// TwinCAT 3 PLC project SuperviserPLC
// ProgramVersion: 3.1.4026.20
// libraries:
//   Tc2_Standard, * (Beckhoff Automation GmbH)
//   Tc2_System, * (Beckhoff Automation GmbH)
//   Tc2_TcpIp, * (Beckhoff Automation GmbH)
//   Tc2_Utilities, * (Beckhoff Automation GmbH)
//   Tc3_EventLogger, * (Beckhoff Automation GmbH)
//   Tc3_JsonXml, * (Beckhoff Automation GmbH)
//   Tc3_Module, * (Beckhoff Automation GmbH)
// project tree:
//   Navitrol Supervisor/Common types/ ST_SectionHeader.TcDUT (not stored), ST_SupervisorHeader.TcDUT
//   Navitrol Supervisor/ FB_Supervisor.TcPOU
//   Navitrol Supervisor/Navitrol to Supervisor response/1100/ ST_1100_Position_initialization_started.TcDUT
//   Navitrol Supervisor/Navitrol to Supervisor response/1101/Components/ E_1101_Initialization_result.TcDUT
//   Navitrol Supervisor/Navitrol to Supervisor response/1101/ ST_1101_Position_initialized.TcDUT (not stored)
//   Navitrol Supervisor/Navitrol to Supervisor response/1126/Components/ ST_1126_Omni_wheels_ref_struct.TcDUT, ST_1126_Supervisor_status_out.TcDUT
//   Navitrol Supervisor/Navitrol to Supervisor response/1126/ ST_1126_Motor_control_omni_response.TcDUT (not stored)
//   Navitrol Supervisor/Navitrol to Supervisor response/3102/Components/ E_3102_Error_status.TcDUT (not stored), E_3102_Position_initialize_status.TcDUT (not stored), E_3102_State.TcDUT (not stored)
//   Navitrol Supervisor/Navitrol to Supervisor response/3102/Components/Sections/1/ ST_3102_1_General_section.TcDUT
//   Navitrol Supervisor/Navitrol to Supervisor response/3102/ ST_3102_Navitrol_status.TcDUT
//   Navitrol Supervisor/Navitrol to Supervisor response/ Param_Supervisor_response.TcGVL (not stored), U_Recived_bytes_from_Navitrol.TcDUT (not stored)
//   Navitrol Supervisor/Supervisor to Navitrol message/1001/ ST_1001_Initialize_position.TcDUT (not stored)
//   Navitrol Supervisor/Supervisor to Navitrol message/1026/Components/ E_1026_Set_drive_mode.TcDUT (not stored), ST_1026_Omni_wheels_struct.TcDUT (not stored), ST_1026_Supervisor_status_bits.TcDUT (not stored)
//   Navitrol Supervisor/Supervisor to Navitrol message/1026/ ST_1026_Measurement_update_generic_omni_drive.TcDUT
//   Navitrol Supervisor/Supervisor to Navitrol message/3002/Components/ E_3002_Set_ESTOP.TcDUT (not stored), E_3002_Status.TcDUT
//   Navitrol Supervisor/Supervisor to Navitrol message/3002/Components/Sections/2/Components/ E_3002_2_Enable_manual_control.TcDUT, E_3002_2_Inactive_Active.TcDUT (not stored)
//   Navitrol Supervisor/Supervisor to Navitrol message/3002/Components/Sections/2/ ST_3002_2_Manual_section.TcDUT (not stored)
//   Navitrol Supervisor/Supervisor to Navitrol message/3002/Components/Sections/6/Components/ E_3002_6_Joystick1_control_mode.TcDUT, E_3002_6_Joystick2_control_mode.TcDUT (not stored), E_3002_6_Steer_type_selection.TcDUT
//   Navitrol Supervisor/Supervisor to Navitrol message/3002/Components/Sections/6/ ST_3002_6_Remote_control_section.TcDUT
//   Navitrol Supervisor/Supervisor to Navitrol message/3002/Components/Sections/8/Components/ ST_3002_8_Binary_data.TcDUT, ST_3002_8_Error_status.TcDUT (not stored)
//   Navitrol Supervisor/Supervisor to Navitrol message/3002/Components/Sections/8/ ST_3002_8_Battery_section.TcDUT
//   Navitrol Supervisor/Supervisor to Navitrol message/3002/Components/Sections/ F_SetSectionHeaderInfo.TcPOU
//   Navitrol Supervisor/Supervisor to Navitrol message/3002/ ST_3002_Supervisor_Status.TcDUT
//   Navitrol Supervisor/Supervisor to Navitrol message/ F_SetHeaderInfo.TcPOU (not stored)
//   / PlcTask.TcTTO
//   POUs/ MAIN.TcPOU
// real-time tasks:
//   TASK PlcTask: cycle T#1ms, priority 20, ADS port 350
// motion (NC):
//   TASK NC-Task 1 SAF: cycle T#2ms, priority 4, ADS port 501
//   TASK NC-Task 1 SVB: cycle T#10ms, priority 8, ADS port 511
//   AXIS LeftWheel (id 1)
//     General: UnitName=m
//     Dynamic: AccelerationMaximum=1, DecelerationMaximum=1, Acceleration=2222, Deceleration=2222, Jerk=224422000
//     Velo: SlowManual=0.6, FastManual=1, Maximum=2.2
//     OtherSettings: AllowMotionCmdToSlave=true
//     encoder EncType=1
//       EncPara: ScaleFactorNumerator=1e-07, EncMode=3
//     drive DrvType=5
//       Analog: VeloReferenz=2.2, TorqueSetpointScale=10, ScaleFactorActTorque=0.1
//       TimeComp: TaskDelayCycles=1
//     controller CtrType=1
//       CtrPara: PriorControlFactor=1
//         Observer: BandWidth=20
//   AXIS RightWheel (id 2)
//     General: UnitName=m
//     Dynamic: AccelerationMaximum=1, DecelerationMaximum=1, Acceleration=2222, Deceleration=2222, Jerk=224422000
//     Velo: SlowManual=0.6, FastManual=1, Maximum=2.2
//     OtherSettings: AllowMotionCmdToSlave=true
//     encoder EncType=1
//       EncPara: ScaleFactorNumerator=1e-07, EncMode=3
//     drive DrvType=5
//       Analog: VeloReferenz=2.2, TorqueSetpointScale=10, ScaleFactorActTorque=0.1
//       TimeComp: TaskDelayCycles=1
//     controller CtrType=1
//       CtrPara: PriorControlFactor=1
//         Observer: BandWidth=20
// variable links:
//   SupervisorPLC Instance <-> NC-Task 1 SAF/Axes/LeftWheel
//     PlcTask Inputs/MAIN.LeftWheel.NcToPlc <-> Outputs/ToPlc
//     PlcTask Outputs/MAIN.LeftWheel.PlcToNc <-> Inputs/FromPlc
//   SupervisorPLC Instance <-> NC-Task 1 SAF/Axes/RightWheel
//     PlcTask Inputs/MAIN.RightWheel.NcToPlc <-> Outputs/ToPlc
//     PlcTask Outputs/MAIN.RightWheel.PlcToNc <-> Inputs/FromPlc

CONFIGURATION SuperviserPLC
    RESOURCE PLC ON TwinCAT3
        TASK PlcTask(INTERVAL := T#1ms, PRIORITY := 20);
        PROGRAM MAIN WITH PlcTask : MAIN;
    END_RESOURCE
END_CONFIGURATION

// ---- Navitrol Supervisor/Common types/ST_SupervisorHeader.TcDUT
{attribute 'pack_mode' := '1'}
{attribute 'hide_all_locals'}
TYPE ST_SupervisorHeader :
	STRUCT
		Protocol_version : UINT;	
		Message_ID		 : UINT;
		Message_length	 : UDINT;
	END_STRUCT
END_TYPE
//When sending a message from Supervisor to Navitrol, this is populated using F_SetHeaderInfo.

// ---- Navitrol Supervisor/Navitrol to Supervisor response/1100/ST_1100_Position_initialization_started.TcDUT
{attribute 'pack_mode' := '1'}
TYPE ST_1100_Position_initialization_started EXTENDS ST_SupervisorHeader :
STRUCT
END_STRUCT
END_TYPE

// ---- Navitrol Supervisor/Navitrol to Supervisor response/1101/Components/E_1101_Initialization_result.TcDUT
{attribute 'qualified_only'}
{attribute 'strict'}
{attribute 'to_string'}
TYPE E_1101_Initialization_result : (
		Failure := 0,
		Success := 1
	) UINT;
END_TYPE
//0 - Failure
//	The position initialization can fail for example if
//		- A good position is not found within pos_ini_max_d..-parameters from the given pos init point
//		- A good position is not found within value of pos_init_max_wait_time-parameter
//		- The AGV is not stationary state, it is performing load or there are scanner related errors active.
//1 - Success
//		- A good position was found near the given position initialization point and position was successfully initialized.

// ---- Navitrol Supervisor/Navitrol to Supervisor response/1126/Components/ST_1126_Omni_wheels_ref_struct.TcDUT
{attribute 'pack_mode' := '1'}
TYPE ST_1126_Omni_wheels_ref_struct :
	STRUCT
		Steer_angle_reference : REAL;
		Wheel_speed_reference : REAL;
	END_STRUCT
END_TYPE

// ---- Navitrol Supervisor/Navitrol to Supervisor response/1126/Components/ST_1126_Supervisor_status_out.TcDUT
{attribute 'pack_mode' := '1'}
TYPE ST_1126_Supervisor_status_out :
	STRUCT
		Navitrol_error : BIT; //	Navitrol has ANY error active AND is unable TO drive.
		Reserved_1	   : BIT;
		Reserved_2	   : BIT;
		Reserved_3	   : BIT;
		Reserved_4	   : BIT;
		Reserved_5	   : BIT;
		Reserved_6	   : BIT;
		Brake_release  : BIT;  //	Navitrol requests Supevisor to release brakes to start driving
		Reserved	   : BYTE; //	Not in use	
	END_STRUCT
END_TYPE

// ---- Navitrol Supervisor/Navitrol to Supervisor response/3102/Components/Sections/1/ST_3102_1_General_section.TcDUT
{attribute 'pack_mode' := '1'}
TYPE ST_3102_1_General_section EXTENDS ST_SectionHeader :
	STRUCT
		Battery_voltage : REAL; // V
		On_route		: UINT; // 1 on route, 0 not on route
	END_STRUCT
END_TYPE

// ---- Navitrol Supervisor/Navitrol to Supervisor response/3102/ST_3102_Navitrol_status.TcDUT
{attribute 'pack_mode' := '1'}
TYPE ST_3102_Navitrol_status EXTENDS ST_SupervisorHeader :
	STRUCT
		DefaultSectionLength	   : UDINT;
		State					   : E_3102_State;
		X_coordinate			   : REAL; //In meters
		Y_coordinate			   : REAL; //In meters
		Heading					   : REAL; //Radians
		Level					   : DINT; //Level ID
		Speed					   : REAL; //m/s
		Position_initialize_status : E_3102_Position_initialize_status;
		Position_confidence		   : UINT; //Position confidence in percentage (1 - 100%)
		Error_status			   : E_3102_Error_status;
		//Additional sections can be added bellow - based on what is requested in the array "Section_IDs" in ST_3002_Supervisor_Status.
		General_section			   : ST_3102_1_General_section;
	END_STRUCT
END_TYPE

// ---- Navitrol Supervisor/Supervisor to Navitrol message/1026/ST_1026_Measurement_update_generic_omni_drive.TcDUT
{attribute 'pack_mode' := '1'}
TYPE ST_1026_Measurement_update_generic_omni_drive EXTENDS ST_SupervisorHeader :
	STRUCT
		Message_number	  : UDINT;
		Set_drive_mode	  : E_1026_Set_drive_mode;
		Supervisor_status : ST_1026_Supervisor_status_bits := (Brake_released := TRUE);
		Number_of_wheels  : UINT						   := 2;
	Omni_wheels: ARRAY [0..1] OF ST_1026_Omni_wheels_struct := [2((Steer_angle := 0.1))];		
	END_STRUCT
END_TYPE

// ---- Navitrol Supervisor/Supervisor to Navitrol message/3002/Components/E_3002_Status.TcDUT
{attribute 'qualified_only'}
{attribute 'strict'}
{attribute 'to_string'}
TYPE E_3002_Status : (
		Not_ok := 0, //ERROR_PLC_FAILURE will be activated, and additionally manual driving will be prevented.
		Ok	   := 1	 //Navitrol is allowed to drive the AGV.
	) UINT;
END_TYPE

// ---- Navitrol Supervisor/Supervisor to Navitrol message/3002/Components/Sections/2/Components/E_3002_2_Enable_manual_control.TcDUT
{attribute 'qualified_only'}
{attribute 'strict'}
{attribute 'to_string'}
TYPE E_3002_2_Enable_manual_control : (
		Enable_control	:= 0,
		Disable_control := 1
	) UINT;
END_TYPE

(*
Used to enable manual control from this section:
	0 - Enable control
Navitrol will activate manual mode and sets WARNING_ETH_MANUAL_MODE. This section can be used to drive the AGV.
	1 - Disable control
Navitrol will ignore any controls from this section.
*)

// ---- Navitrol Supervisor/Supervisor to Navitrol message/3002/Components/Sections/6/Components/E_3002_6_Joystick1_control_mode.TcDUT
{attribute 'qualified_only'}
{attribute 'strict'}
{attribute 'to_string'}
TYPE E_3002_6_Joystick1_control_mode : (
		No_control	   := 0,
		Old_control	   := 1,
		Vector_control := 2
	)UINT;
END_TYPE

(*
Selects the joystick 1 control mode:
	0 - No control
Joystick 1 x and y values are ignored.
	1 - Old control
	Not recommended
	Navitrol activates manual mode. Curvature is calculated directly from joystick 1 x value and the speed from joystick 1 y value.
2 - Vector control
	Recommended
	Navitrol activates manual mode. A unit vector is calculated from joystick 1 xy-values. The speed comes from the length of the vector (Positive when y is positive) and the curvature from its angle from the Y-axis.
	For example AGV drives forward and curves right when x and y are positive.
	For more information, see "Joystick System" chapter from Web Interface document

*)

// ---- Navitrol Supervisor/Supervisor to Navitrol message/3002/Components/Sections/6/Components/E_3002_6_Steer_type_selection.TcDUT
{attribute 'qualified_only'}
{attribute 'strict'}
{attribute 'to_string'}
TYPE E_3002_6_Steer_type_selection : (
		Invalid					:= 0,
		Front_wheel_steer		:= 1,
		Mid_wheel_steer			:= 2,
		Rear_wheel_steer		:= 3,
		Pivot_steer				:= 5,
		Parallel_steer_forward	:= 6,
		Parallel_steer_backward := 7
	);
END_TYPE

(*
1 - Front wheel steer
Only for omni drives. Moves the navigation point to between the front wheels. With this steer type almost all turning control will be done by the rear wheels.
2 - Mid wheel steer
	Normal driving. The normal navigation point is used.
3 - Rear wheel steer
	Only for omni drives. Moves the navigation point to between the rear wheels. With this steer type almost all turning control will be done by the front wheels.
5 - Pivot steer
	Pivot curvature is always given, and supervisor can control only the speed up to maximum of pivot_speed-parameter. This mode should only be activated, if the AGV can pivot.
6 - Parallel steer forward
	Only for omni drives.
	The curvature in this mode is always zero. Instead of curvature supervisor controls the frame heading instead and speed. Wheels will rotate forward with positive speed reference.
7 - Parallel steer backward
	Only for omni drives.
	The curvature in this mode is always zero. Instead of curvature supervisor controls the frame heading instead and speed. Wheels will rotate backwards with positive speed reference.

*)

// ---- Navitrol Supervisor/Supervisor to Navitrol message/3002/Components/Sections/6/ST_3002_6_Remote_control_section.TcDUT
{attribute 'pack_mode' := '1'}
TYPE ST_3002_6_Remote_control_section EXTENDS ST_SectionHeader :
	STRUCT
		Joystick1_control_mode : E_3002_6_Joystick1_control_mode;
		Joystick1_x			   : REAL;
		Joystick1_y			   : REAL;
		Joystick2_control_mode : E_3002_6_Joystick2_control_mode;
		Joystick2_x			   : REAL; //0 - Not in use
		Joystick2_y			   : REAL; (*Lift actuator height reference control.
										If the given y-value is larger than 0.1 actuator control is enabled. 
										And the y-value is scaled with actuator_eth_ctrl_scale-parameter and added to the previous actuator reference. 
										The actuator reference can be controlled only between values of actuator_min_val and actuator_max_val parameters.Valid values [-1...1]*)
		Steer_type_selection : E_3002_6_Steer_type_selection;
	END_STRUCT
END_TYPE

// ---- Navitrol Supervisor/Supervisor to Navitrol message/3002/Components/Sections/8/Components/ST_3002_8_Binary_data.TcDUT
{attribute 'pack_mode' := '1'}
TYPE ST_3002_8_Binary_data :
STRUCT
	Request_charge   : BIT; // This charge request info is show in motor control messages and in Navitrol battery status section if charging_cmd_source-parameter is set to 3. No drive orders or other actions are made based on this.
	Charging_active  : BIT; // Informs Navitrol that charging is active. Navitrol will set soft stop (parameter charging_prevents_driving).
	Balancing_active : BIT; // Informs Navitrol that battery balancing is active at charger. Navitrol will set soft stop (parameter charging_prevents_driving).
	Reserved_3       : BIT; // 0 - Not in use
	Reserved_4       : BIT; // 0 - Not in use
	Reserved_5       : BIT; // 0 - Not in use
	Reserved_6       : BIT; // 0 - Not in use
	Reserved_7       : BIT; // 0 - Not in use
END_STRUCT
END_TYPE

// ---- Navitrol Supervisor/Supervisor to Navitrol message/3002/Components/Sections/8/ST_3002_8_Battery_section.TcDUT
{attribute 'pack_mode' := '1'}
TYPE ST_3002_8_Battery_section EXTENDS ST_SectionHeader :
	STRUCT
		// Battery state of charge percentage. Valid values [0...100] 65535 - Not available

		// This will be used for determining the battery level if battery_percentage_from_mot_ctrl-parameter is set to 1.
		State_of_charge : UINT := 100;
		// Battery voltage in 0.1 Volts. For example, 4.2V would be 42 65535 - Not available

		// This will be used for determining the battery level if battery_percentage_from_mot_ctrl-parameter is set to 0.
		Voltage : UINT := 42;
		// Charge current / current draw in 0.1 Amperes. Negative values when battery is discharging

		// and positive values when battery is being charged. 32767 - Not available

		// Only for statistics - visible in Navitrol Monitor.
		Charge_current_draw : INT := 10;
		// Energy draw in 0.1 Ampere hours Negative values when battery is discharging

		// and positive values when battery is being charged. 32767 - Not available

		// Only for statistics - visible in Navitrol Monitor.
		Energy_draw : INT := 100;
		// Estimated time left in minutes until the battery is empty. 65535 - Not available

		// Only for statistics - visible in Navitrol Monitor.
		Time_remaining : UINT := 45;
		// Battery state of health percentage. Describes the overall state of the battery. Valid values [0...100] 65535 - Not available

		// Only for statistics - visible in Navitrol Monitor.
		State_of_health : UINT := 100;
		// Battery temperature in Celsius degrees. 32767 - Not available

		// Used to trigger WARNING_BATTERY_HIGH_TEMPERATURE if given temperature is larger than

		// battery_high_temperature_warning_limit_C and ERROR_BATTERY_HIGH_TEMPERATURE if larger

		// than battery_high_temperature_error_limit_C
		Temperature : INT := 32;
		// Total number of load cycles performed for the battery. 65535 - Not available

		// Only for statistics - visible in Navitrol Monitor.
		Load_cycle_count : UINT := 20;
		// Total number of operating hours of the battery. 65535 - Not available

		// Only for statistics - visible in Navitrol Monitor.
		Operating_hours : UINT := 155;
		// Voltage of the charger in 0.1 Volts. 65535 - Not available

		// Only for statistics - visible in Navitrol Monitor.
		Charger_voltage : UINT := 420;
		// Error status information. If any of the errors marked with * are active Navitrol Monitor will view its description

		// and Navitrol set WARNING_BATTERY_ERROR_OR_WARNING_ACTIVE 0 - No error
		Error_status : ST_3002_8_Error_status;
		// Battery related binary data and requests 0 - Inactive
		Binary_data : ST_3002_8_Binary_data;
		// 0 - Not in use
		Reserved : BYTE;
	END_STRUCT
END_TYPE

// ---- Navitrol Supervisor/Supervisor to Navitrol message/3002/ST_3002_Supervisor_Status.TcDUT
{attribute 'pack_mode' := '1'}
TYPE ST_3002_Supervisor_Status EXTENDS ST_SupervisorHeader :
	STRUCT
		Status			   : E_3002_Status := E_3002_Status.Ok;
		Set_Estop		   : E_3002_Set_ESTOP;
		Number_of_sections : UINT				 := 1;	 //Number of sections requested in response message 3102 - Needs to be the same number as the array size Section_IDs. if 0 - then Section_IDs can be commented out
		Section_IDs		   : ARRAY[0..0] OF UINT := [1]; //List of sections to send in the response message 3102
		Manual_section: ST_3002_2_Manual_section := (Enable_manual_control := E_3002_2_Enable_manual_control.Disable_control);		
		Battery_section	   : ST_3002_8_Battery_section;
	END_STRUCT
END_TYPE

// ---- POUs/MAIN.TcPOU
PROGRAM MAIN
VAR
	Supervisor				 : FB_Supervisor := (RemoteHost := '127.0.0.1', RemotePort := 2000);
END_VAR

Supervisor(Execute := TRUE);

END_PROGRAM

// ---- Navitrol Supervisor/FB_Supervisor.TcPOU
FUNCTION_BLOCK FB_Supervisor
VAR_INPUT
	RemoteHost									 : T_IPv4Addr := '127.0.0.1';
	RemotePort									 : UDINT	  := 2000;	  //Needs to match Navitrol parameter "supervisor_eth_port"
	CycleTime3002								 : TIME		  := T#100MS; //maximum interval 1 second
	CycleTime1026								 : TIME		  := T#30MS;  //This needs to match the Navitrol parameter "control_interval_us"
	Execute										 : BOOL;				  //Connect to Navitrol, and establish comuncations. If false, the socket is closed.
	st3002_Supervisor_Status					 : ST_3002_Supervisor_Status;
	st1026_Measurement_update_generic_omni_drive : ST_1026_Measurement_update_generic_omni_drive;
	Initialize_position							 : BOOL; //Rising edge trigger to send a Initialize position command 
	st1001_Initialize_position					 : ST_1001_Initialize_position := (X := 100.0, Y := 150.0);
END_VAR

VAR_OUTPUT
	st3102_Navitrol_status			   : ST_3102_Navitrol_status;
	st1126_Motor_control_omni_response : ST_1126_Motor_control_omni_response;
	st1101_Position_initialized		   : ST_1101_Position_initialized;
	Busy							   : BOOL;
	Error							   : BOOL;
	ErrorID							   : UDINT;
END_VAR

VAR
	State : (INIT_FBs,
		CLOSE_OLD_SOCKETS,
		CONNECT_TO_Server,
		COMS_ACTIVE,
		CLOSE_CONNECTION);
	CloseAll : FB_SocketCloseAll;
	Connect	 : FB_SocketConnect;
	Close	 : FB_SocketClose;

	//Event logging
	FirstScan  : BOOL := TRUE;
	ErrorMsg   : FB_TcMessage;
	WarnMsg	   : FB_TcMessage;
	VerboseMsg : FB_TcMessage;
END_VAR

IF FirstScan THEN
	ErrorMsg.CreateEx(stEventEntry := TC_EVENTS.TcpIpComms.ErrorMsg, ipSourceInfo := 0);
	VerboseMsg.CreateEx(stEventEntry := TC_EVENTS.TcpIpComms.VerboseMsg, ipSourceInfo := 0);
	WarnMsg.CreateEx(stEventEntry := TC_EVENTS.TcpIpComms.WarnMsg, ipSourceInfo := 0);
	FirstScan := FALSE;
END_IF

CASE State OF
	INIT_FBs:
		CloseAll(bExecute := FALSE);
		Connect(bExecute := FALSE);
		Close(bExecute := FALSE);
		Busy := FALSE;
		IF Execute THEN
			Busy := TRUE;
			IF CycleTime3002 = T#0S OR CycleTime3002 > T#1S THEN
				ErrorMsg.ipArguments.Clear().AddString('Invalid input CycleTime3002');
				ErrorMsg.Send();
				Error := TRUE;
				RETURN;
			END_IF

			State := CLOSE_OLD_SOCKETS;
			Error := FALSE;
			VerboseMsg.ipArguments.Clear().AddString('Starting communications to:').AddString(RemoteHost).AddUDInt(RemotePort);
			VerboseMsg.Send();
		END_IF

	CLOSE_OLD_SOCKETS: //In the event of online change or download
		CloseAll(sSrvNetId := '', bExecute := TRUE, tTimeout := T#10S);
		IF NOT CloseAll.bBusy THEN
			CloseAll(bExecute := FALSE);
			State := CONNECT_TO_Server;
		END_IF

	CONNECT_TO_Server:
		Connect(sSrvNetId	:= '',
				sRemoteHost := RemoteHost,
				nRemotePort := RemotePort,
				bExecute	:= TRUE,
				tTimeout	:= T#4S);

		IF NOT Connect.bBusy THEN
			IF NOT Connect.bError THEN
				IF Connect.hSocket.handle <> 0 THEN
					State := COMS_ACTIVE;
					VerboseMsg.ipArguments.Clear().AddString('Connected to server:').AddString(RemoteHost).AddUDInt(RemotePort).AddString('Local port').AddUDInt(Connect.hSocket.localAddr.nPort);
					VerboseMsg.Send();
				END_IF
			ELSE
				Error := TRUE;
				State := INIT_FBs;
				ErrorMsg.ipArguments.Clear().AddString('Failed to connect to server:').AddString(RemoteHost).AddUDInt(RemotePort).AddString(', Error:').AddUDInt(Connect.nErrId);
				ErrorMsg.Send();
			END_IF

			Connect(bExecute := FALSE);
		END_IF

	COMS_ACTIVE:
		SendMsg3002();
		SendMsg1026();
		SendMsg1001();
		ReciveAllMsgsAndParse();
		IF NOT Execute THEN
			VerboseMsg.ipArguments.Clear().AddString('Connection closed by user');
			VerboseMsg.Send();
			State := CLOSE_CONNECTION;
		END_IF

	CLOSE_CONNECTION:
		Close(sSrvNetId := '',
			  hSocket	:= Connect.hSocket,
			  bExecute	:= TRUE,
			  tTimeout	:= T#4S);

		IF NOT Close.bBusy THEN
			Close(bExecute := FALSE);
			State := INIT_FBs;
		END_IF
END_CASE

METHOD INTERNAL ReciveAllMsgsAndParse : HRESULT
VAR_INST
	Receive								   : FB_SocketReceive;
	ReceiveBuffer						   : U_Recived_bytes_from_Navitrol;
	NumOf1100MsgRecived					   : UDINT;
	st1100_Position_initialization_started : ST_1100_Position_initialization_started;
	NumOf1101MsgRecived					   : UDINT;
	NumOf3102MsgRecived					   : UDINT;
	NumOf1126MsgRecived					   : UDINT;
	UnknowMsgRecivedCounter				   : UDINT;
	UnknowMsg							   : U_Recived_bytes_from_Navitrol;
END_VAR
Receive(sSrvNetId := '',
		hSocket	  := Connect.hSocket,
		cbLen	  := SIZEOF(ReceiveBuffer),
		pDest	  := ADR(ReceiveBuffer),
		bExecute  := TRUE,
		tTimeout  := T#10S);

IF NOT Receive.bBusy THEN
	IF Receive.nRecBytes <> 0 THEN
		IF Receive.nRecBytes = SIZEOF(ReceiveBuffer) THEN
			ErrorMsg.ipArguments.Clear().AddString('Recive buffer is not large enough! Please increase the size of "Param_Supervisor_response.RecivedBytesBufferSize');
			ErrorMsg.Send();
			State	:= CLOSE_CONNECTION;
			Error	:= TRUE;
			ErrorID := Global.TC_EVENTS.TcGeneralAdsEventClass.NoMemory.nEventId;
			RETURN;
		END_IF

		CASE ReceiveBuffer.Header.Message_ID OF //Check what message type is being recived - then copy it into the correct structure
			1100:
				NumOf1100MsgRecived := NumOf1100MsgRecived + 1;
				MEMCPY(destAddr := ADR(st1100_Position_initialization_started), srcAddr := ADR(ReceiveBuffer), n := SIZEOF(st1100_Position_initialization_started));
				VerboseMsg.ipArguments.Clear().AddString('Position initialization started');
				VerboseMsg.Send();

			1101:
				NumOf1101MsgRecived := NumOf1101MsgRecived + 1;
				MEMCPY(destAddr := ADR(st1101_Position_initialized), srcAddr := ADR(ReceiveBuffer), n := SIZEOF(st1101_Position_initialized));
				VerboseMsg.ipArguments.Clear().AddString('Position initialization finished');
				VerboseMsg.Send();

			1126:
				NumOf1126MsgRecived := NumOf1126MsgRecived + 1;
				MEMCPY(destAddr := ADR(st1126_Motor_control_omni_response), srcAddr := ADR(ReceiveBuffer), n := SIZEOF(st1126_Motor_control_omni_response));

			3102:
				NumOf3102MsgRecived := NumOf3102MsgRecived + 1;
				MEMCPY(destAddr := ADR(st3102_Navitrol_status), srcAddr := ADR(ReceiveBuffer), n := SIZEOF(st3102_Navitrol_status));

		ELSE
			UnknowMsgRecivedCounter := UnknowMsgRecivedCounter + 1;
			MEMCPY(destAddr := ADR(UnknowMsg), srcAddr := ADR(ReceiveBuffer), n := SIZEOF(UnknowMsg));
			WarnMsg.ipArguments.Clear().AddString('Unknow msg type recived with ID:').AddUInt(ReceiveBuffer.Header.Message_ID).AddString('Contents:').AddBlob(pData := ADR(ReceiveBuffer), cbData := TO_UINT(Receive.nRecBytes));
			WarnMsg.Send();
		END_CASE
	END_IF

	Receive(bExecute := FALSE);

	//Clear recive buffer
	MEMSET(destAddr := ADR(ReceiveBuffer), fillByte := 0, n := SIZEOF(ReceiveBuffer));
END_IF

IF Receive.bError THEN
	ErrorMsg.ipArguments.Clear().AddString('Failed to Receive, Error:').AddUDInt(Receive.nErrId);
	ErrorMsg.Send();
	State	:= CLOSE_CONNECTION;
	Error	:= TRUE;
	ErrorID := Receive.nErrId;
END_IF
END_METHOD

METHOD INTERNAL SendMsg1001 : HRESULT
VAR_INST
	rtInitialize_position : R_TRIG;
	Send1001			  : FB_SocketSend;
END_VAR
rtInitialize_position(CLK := Initialize_position);
IF rtInitialize_position.Q THEN
	F_SetHeaderInfo(st1001_Initialize_position);
	MEMSET(destAddr := ADR(st1101_Position_initialized), fillByte := 0, n := SIZEOF(st1101_Position_initialized)); //Clear old results
END_IF

Send1001(sSrvNetId := '',
		 hSocket   := Connect.hSocket,
		 cbLen	   := SIZEOF(st1001_Initialize_position),
		 pSrc	   := ADR(st1001_Initialize_position),
		 bExecute  := rtInitialize_position.Q,
		 tTimeout  := T#2S);

IF Send1001.bError THEN
	ErrorMsg.ipArguments.Clear().AddString('Failed to send 1001 Error:').AddUDInt(Send1001.nErrId);
	ErrorMsg.Send();
END_IF
END_METHOD

METHOD INTERNAL SendMsg1026 : HRESULT
VAR_INST
	Timer1026 : TON;
	Send1026  : FB_SocketSend;
END_VAR
Timer1026(IN := NOT Timer1026.Q, PT := CycleTime1026);
IF Timer1026.Q THEN
	F_SetHeaderInfo(st1026_Measurement_update_generic_omni_drive);
	st1026_Measurement_update_generic_omni_drive.Message_number := st1026_Measurement_update_generic_omni_drive.Message_number + 1;
END_IF

Send1026(sSrvNetId := '',
		 hSocket   := Connect.hSocket,
		 cbLen	   := SIZEOF(st1026_Measurement_update_generic_omni_drive),
		 pSrc	   := ADR(st1026_Measurement_update_generic_omni_drive),
		 bExecute  := Timer1026.Q,
		 tTimeout  := T#2S);

IF Send1026.bError THEN
	ErrorMsg.ipArguments.Clear().AddString('Failed to send 1026 Error:').AddUDInt(Send1026.nErrId);
	ErrorMsg.Send();
	State	:= CLOSE_CONNECTION;
	Error	:= TRUE;
	ErrorID := Send1026.nErrId;
END_IF
END_METHOD

METHOD INTERNAL SendMsg3002 : HRESULT
VAR_INST
	Timer3002 : TON;
	Send3002  : FB_SocketSend;
END_VAR
Timer3002(IN := NOT Timer3002.Q, PT := CycleTime3002);
IF Timer3002.Q THEN
	F_SetHeaderInfo(st3002_Supervisor_Status);
	F_SetSectionHeaderInfo(st3002_Supervisor_Status.Manual_section);
	F_SetSectionHeaderInfo(st3002_Supervisor_Status.Battery_section);
	//Populate any added section headers here
END_IF

Send3002(sSrvNetId := '',
		 hSocket   := Connect.hSocket,
		 cbLen	   := SIZEOF(st3002_Supervisor_Status),
		 pSrc	   := ADR(st3002_Supervisor_Status),
		 bExecute  := Timer3002.Q,
		 tTimeout  := T#2S);

IF Send3002.bError THEN
	ErrorMsg.ipArguments.Clear().AddString('Failed to send 3002 Error:').AddUDInt(Send3002.nErrId);
	ErrorMsg.Send();
	State	:= CLOSE_CONNECTION;
	Error	:= TRUE;
	ErrorID := Send3002.nErrId;
END_IF
END_METHOD

END_FUNCTION_BLOCK

// ---- Navitrol Supervisor/Supervisor to Navitrol message/3002/Components/Sections/F_SetSectionHeaderInfo.TcPOU
FUNCTION F_SetSectionHeaderInfo : HRESULT
VAR_INPUT
	Section : ANY;
END_VAR

VAR
	SectionHeader		  : ST_SectionHeader;
	fbJsonDataType		  : FB_JsonReadWriteDataType;
	DataTypeName		  : STRING;
	Message_ID			  : UINT;
	GetDataTypeNameResult : HRESULT;
	i					  : INT;
	StartPos			  : INT;
	EndPos				  : INT;
	IDString			  : STRING;
	ParseSuccess		  : BOOL;
END_VAR

IF Section.diSize < 0 THEN
	F_SetSectionHeaderInfo := S_FALSE;
	RETURN;
END_IF

DataTypeName := fbJsonDataType.GetDataTypeNameByAddress(nData := TO_UDINT(Section.diSize), pData := Section.pValue, hrErrorCode => GetDataTypeNameResult);

// Parse Message_ID from DataTypeName (e.g., 'ST_3002_2_Manual_section' -> 2)
ParseSuccess := FALSE;
StartPos	 := FIND(DataTypeName, 'ST_3002_');
IF StartPos > 0 THEN
	StartPos := StartPos + 8; // Move past 'ST_3002_'

	// Find the next underscore after the ID
	EndPos := 0;
	FOR i := StartPos TO LEN(DataTypeName) DO
		IF MID(DataTypeName, 1, i) = '_' THEN
			EndPos := i;
			EXIT;
		END_IF
	END_FOR

	IF EndPos > StartPos THEN
		// Extract the ID substring
		IDString	 := MID(DataTypeName, EndPos - StartPos, StartPos);
		Message_ID	 := STRING_TO_UINT(IDString);
		ParseSuccess := TRUE;
	END_IF
END_IF

// Fallback if parsing fails
IF NOT ParseSuccess THEN
	Message_ID		:= 0;
	F_SetSectionHeaderInfo := S_FALSE;
	RETURN;
END_IF

// All 3002 messages sections start with ST_SectionHeader
SectionHeader.Section_ID:=Message_ID;
SectionHeader.Section_length:=TO_UDINT(Section.diSize);


// Copy populated header into Section
MEMCPY(destAddr := Section.pValue, srcAddr := ADR(SectionHeader), n := SIZEOF(SectionHeader));
F_SetSectionHeaderInfo := S_OK;

END_FUNCTION
